// TIA Portal V17 export
// export: Created 2025-06-26T06:49:10.1287295Z, ExportSetting WithDefaults, DisplayName Totally Integrated Automation Portal, DisplayVersion V17 Update 8, DisplayName TIA Portal Openness, DisplayVersion V17 Update 8, DisplayName TIA Portal Version Control Interface, DisplayVersion V17, DisplayName STEP 7 Professional, DisplayVersion V17 Update 8, DisplayName STEP 7 Safety, DisplayVersion V17 Update 6, DisplayName WinCC Advanced, DisplayVersion V17 Update 8
FUNCTION_BLOCK "AnalogInputProcessing"   // FB37, FBD
TITLE = Handle analog inputs
{ S7_Optimized_Access := 'TRUE' }
AUTHOR : Heaten
VERSION : 0.1
// Map & scale analog inputs
// stored: AutoNumber true, IsIECCheckEnabled false, IsRetainMemResEnabled false, MemoryReserve 0, SetENOAutomatically false, UDAEnableTagReadback false
   VAR
      bHere : Bool;
   END_VAR
   VAR_TEMP
      fDummy : Real;
      fMaxWindingTemperature : Real;
      HBL_PT_05 : Real;
   END_VAR
   VAR_TEMP   // added for the SCL form of the ladder/FBD networks
      _w1 : Bool;
   END_VAR
BEGIN

REGION Network 1: HBL_TT_03 Oil sump oil temperature
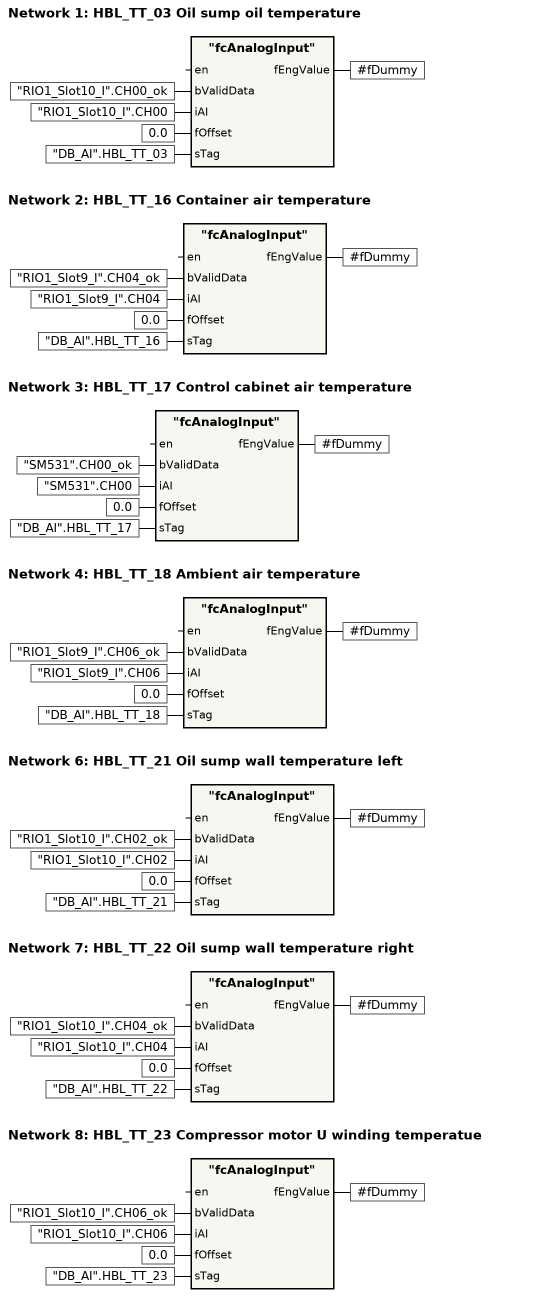
   "fcAnalogInput"(bValidData := "RIO1_Slot10_I".CH00_ok,
                   iAI := "RIO1_Slot10_I".CH00,
                   fOffset := 0.0,
                   sTag := "DB_AI".HBL_TT_03,
                   fEngValue => #fDummy);
END_REGION

REGION Network 2: HBL_TT_16 Container air temperature
   "fcAnalogInput"(bValidData := "RIO1_Slot9_I".CH04_ok,
                   iAI := "RIO1_Slot9_I".CH04,
                   fOffset := 0.0,
                   sTag := "DB_AI".HBL_TT_16,
                   fEngValue => #fDummy);
END_REGION

REGION Network 3: HBL_TT_17 Control cabinet air temperature
   "fcAnalogInput"(bValidData := "SM531".CH00_ok,
                   iAI := "SM531".CH00,
                   fOffset := 0.0,
                   sTag := "DB_AI".HBL_TT_17,
                   fEngValue => #fDummy);
END_REGION

REGION Network 4: HBL_TT_18 Ambient air temperature
   "fcAnalogInput"(bValidData := "RIO1_Slot9_I".CH06_ok,
                   iAI := "RIO1_Slot9_I".CH06,
                   fOffset := 0.0,
                   sTag := "DB_AI".HBL_TT_18,
                   fEngValue => #fDummy);
END_REGION

REGION Network 5: HBL_TT_19 Main inverter temperature
   // ##This is a fieldbus value. get from inverter, if we need it.
END_REGION

REGION Network 6: HBL_TT_21 Oil sump wall temperature left
   "fcAnalogInput"(bValidData := "RIO1_Slot10_I".CH02_ok,
                   iAI := "RIO1_Slot10_I".CH02,
                   fOffset := 0.0,
                   sTag := "DB_AI".HBL_TT_21,
                   fEngValue => #fDummy);
END_REGION

REGION Network 7: HBL_TT_22 Oil sump wall temperature right
   "fcAnalogInput"(bValidData := "RIO1_Slot10_I".CH04_ok,
                   iAI := "RIO1_Slot10_I".CH04,
                   fOffset := 0.0,
                   sTag := "DB_AI".HBL_TT_22,
                   fEngValue => #fDummy);
END_REGION

REGION Network 8: HBL_TT_23 Compressor motor U winding temperatue
   "fcAnalogInput"(bValidData := "RIO1_Slot10_I".CH06_ok,
                   iAI := "RIO1_Slot10_I".CH06,
                   fOffset := 0.0,
                   sTag := "DB_AI".HBL_TT_23,
                   fEngValue => #fDummy);
END_REGION

REGION Network 9: HBL_TT_24 Compressor motor V winding temperature
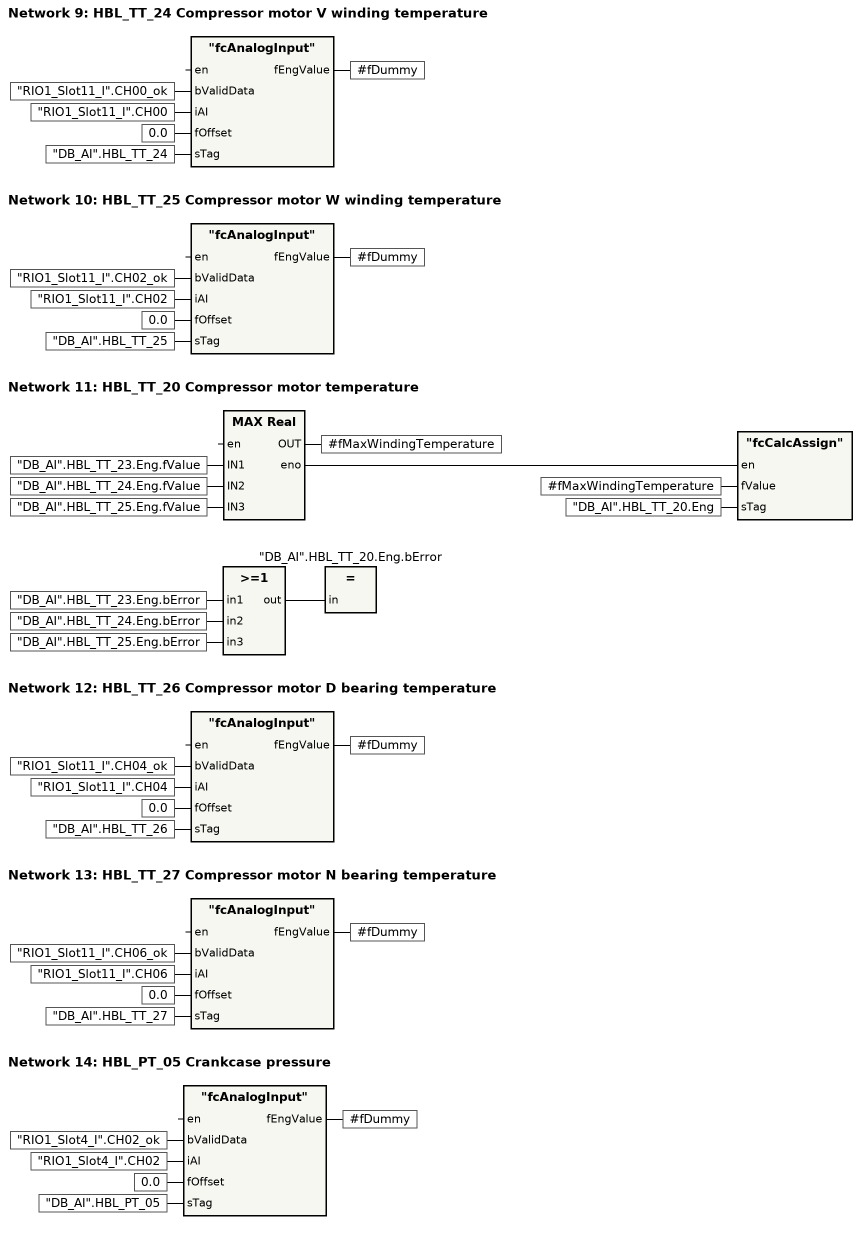
   "fcAnalogInput"(bValidData := "RIO1_Slot11_I".CH00_ok,
                   iAI := "RIO1_Slot11_I".CH00,
                   fOffset := 0.0,
                   sTag := "DB_AI".HBL_TT_24,
                   fEngValue => #fDummy);
END_REGION

REGION Network 10: HBL_TT_25 Compressor motor W winding temperature
   "fcAnalogInput"(bValidData := "RIO1_Slot11_I".CH02_ok,
                   iAI := "RIO1_Slot11_I".CH02,
                   fOffset := 0.0,
                   sTag := "DB_AI".HBL_TT_25,
                   fEngValue => #fDummy);
END_REGION

REGION Network 11: HBL_TT_20 Compressor motor temperature
   // MAX of any of the winding temperatures. If there is only one motor temperature, eg one PTC, use HBL-TT-20 as the analog input object
   // The individual winding temperatures are not used in the program (but are available for monitoring & logging)
   #fMaxWindingTemperature := MAX(IN1 := "DB_AI".HBL_TT_23.Eng.fValue, IN2 := "DB_AI".HBL_TT_24.Eng.fValue, IN3 := "DB_AI".HBL_TT_25.Eng.fValue);
   "fcCalcAssign"(fValue := #fMaxWindingTemperature, sTag := "DB_AI".HBL_TT_20.Eng);
   "DB_AI".HBL_TT_20.Eng.bError := "DB_AI".HBL_TT_23.Eng.bError OR "DB_AI".HBL_TT_24.Eng.bError OR "DB_AI".HBL_TT_25.Eng.bError;
END_REGION

REGION Network 12: HBL_TT_26 Compressor motor D bearing temperature
   "fcAnalogInput"(bValidData := "RIO1_Slot11_I".CH04_ok,
                   iAI := "RIO1_Slot11_I".CH04,
                   fOffset := 0.0,
                   sTag := "DB_AI".HBL_TT_26,
                   fEngValue => #fDummy);
END_REGION

REGION Network 13: HBL_TT_27 Compressor motor N bearing temperature
   "fcAnalogInput"(bValidData := "RIO1_Slot11_I".CH06_ok,
                   iAI := "RIO1_Slot11_I".CH06,
                   fOffset := 0.0,
                   sTag := "DB_AI".HBL_TT_27,
                   fEngValue => #fDummy);
END_REGION

REGION Network 14: HBL_PT_05 Crankcase pressure
   "fcAnalogInput"(bValidData := "RIO1_Slot4_I".CH02_ok,
                   iAI := "RIO1_Slot4_I".CH02,
                   fOffset := 0.0,
                   sTag := "DB_AI".HBL_PT_05,
                   fEngValue => #fDummy);
END_REGION

REGION Network 15: HBL_CT_01 Gas detector
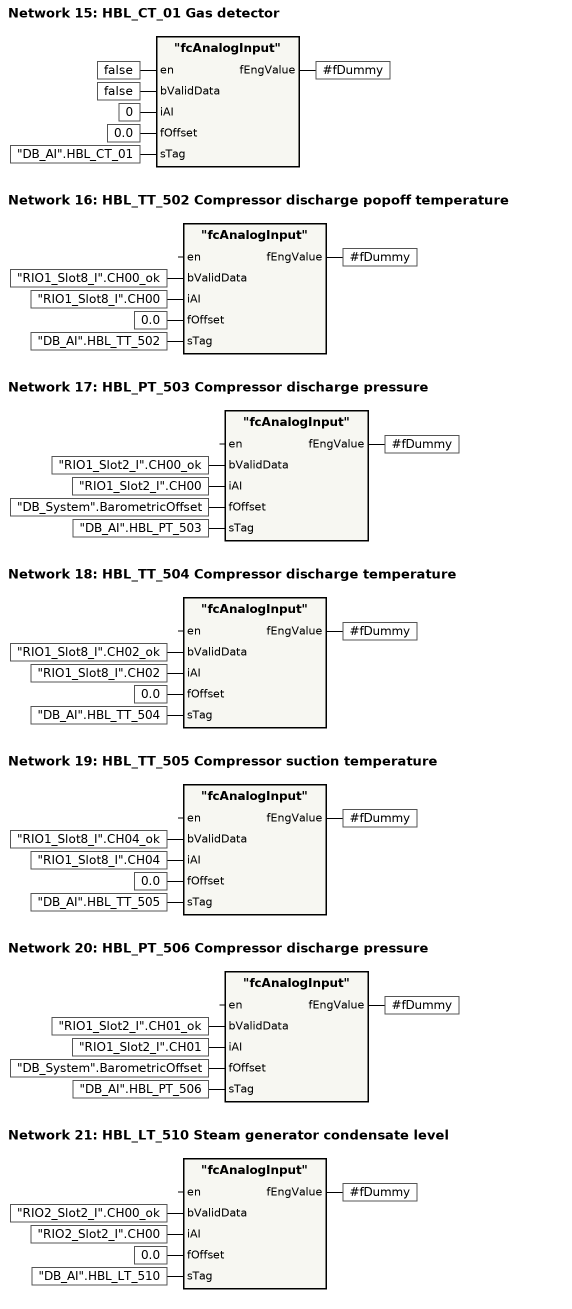
   IF false THEN
       "fcAnalogInput"(bValidData := false,
                       iAI := 0,
                       fOffset := 0.0,
                       sTag := "DB_AI".HBL_CT_01,
                       fEngValue => #fDummy);
   END_IF;
END_REGION

REGION Network 16: HBL_TT_502 Compressor discharge popoff temperature
   "fcAnalogInput"(bValidData := "RIO1_Slot8_I".CH00_ok,
                   iAI := "RIO1_Slot8_I".CH00,
                   fOffset := 0.0,
                   sTag := "DB_AI".HBL_TT_502,
                   fEngValue => #fDummy);
END_REGION

REGION Network 17: HBL_PT_503 Compressor discharge pressure
   "fcAnalogInput"(bValidData := "RIO1_Slot2_I".CH00_ok,
                   iAI := "RIO1_Slot2_I".CH00,
                   fOffset := "DB_System".BarometricOffset,
                   sTag := "DB_AI".HBL_PT_503,
                   fEngValue => #fDummy);
END_REGION

REGION Network 18: HBL_TT_504 Compressor discharge temperature
   "fcAnalogInput"(bValidData := "RIO1_Slot8_I".CH02_ok,
                   iAI := "RIO1_Slot8_I".CH02,
                   fOffset := 0.0,
                   sTag := "DB_AI".HBL_TT_504,
                   fEngValue => #fDummy);
END_REGION

REGION Network 19: HBL_TT_505 Compressor suction temperature
   "fcAnalogInput"(bValidData := "RIO1_Slot8_I".CH04_ok,
                   iAI := "RIO1_Slot8_I".CH04,
                   fOffset := 0.0,
                   sTag := "DB_AI".HBL_TT_505,
                   fEngValue => #fDummy);
END_REGION

REGION Network 20: HBL_PT_506 Compressor discharge pressure
   "fcAnalogInput"(bValidData := "RIO1_Slot2_I".CH01_ok,
                   iAI := "RIO1_Slot2_I".CH01,
                   fOffset := "DB_System".BarometricOffset,
                   sTag := "DB_AI".HBL_PT_506,
                   fEngValue => #fDummy);
END_REGION

REGION Network 21: HBL_LT_510 Steam generator condensate level
   "fcAnalogInput"(bValidData := "RIO2_Slot2_I".CH00_ok,
                   iAI := "RIO2_Slot2_I".CH00,
                   fOffset := 0.0,
                   sTag := "DB_AI".HBL_LT_510,
                   fEngValue => #fDummy);
END_REGION

REGION Network 22: HBL_PT_511 Heat sink discharge pressure
   // Local or remote
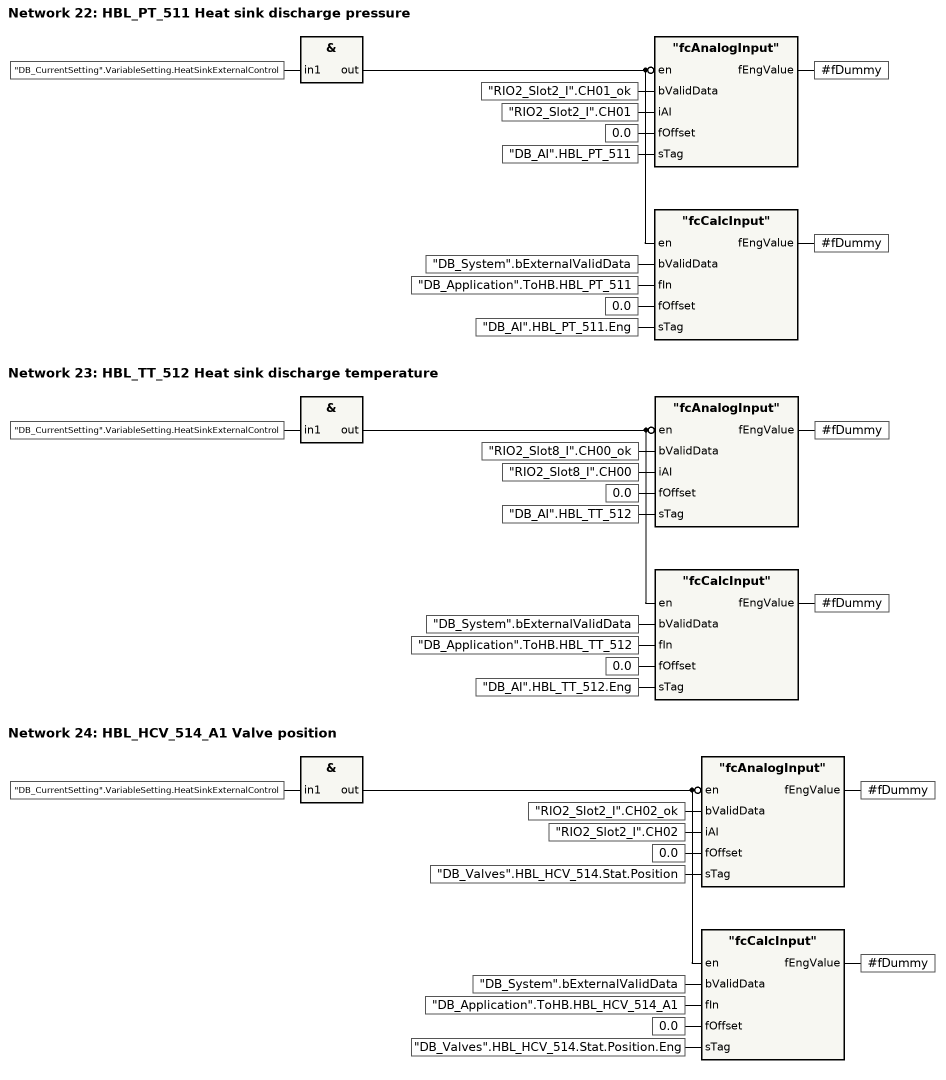
   #_w1 := "DB_CurrentSetting".VariableSetting.HeatSinkExternalControl;
   IF NOT "DB_CurrentSetting".VariableSetting.HeatSinkExternalControl THEN
       "fcAnalogInput"(bValidData := "RIO2_Slot2_I".CH01_ok,
                       iAI := "RIO2_Slot2_I".CH01,
                       fOffset := 0.0,
                       sTag := "DB_AI".HBL_PT_511,
                       fEngValue => #fDummy);
   END_IF;
   IF #_w1 THEN
       "fcCalcInput"(bValidData := "DB_System".bExternalValidData,
                     fIn := "DB_Application".ToHB.HBL_PT_511,
                     fOffset := 0.0,
                     sTag := "DB_AI".HBL_PT_511.Eng,
                     fEngValue => #fDummy);
   END_IF;
END_REGION

REGION Network 23: HBL_TT_512 Heat sink discharge temperature
   // Local or remote
   #_w1 := "DB_CurrentSetting".VariableSetting.HeatSinkExternalControl;
   IF NOT "DB_CurrentSetting".VariableSetting.HeatSinkExternalControl THEN
       "fcAnalogInput"(bValidData := "RIO2_Slot8_I".CH00_ok,
                       iAI := "RIO2_Slot8_I".CH00,
                       fOffset := 0.0,
                       sTag := "DB_AI".HBL_TT_512,
                       fEngValue => #fDummy);
   END_IF;
   IF #_w1 THEN
       "fcCalcInput"(bValidData := "DB_System".bExternalValidData,
                     fIn := "DB_Application".ToHB.HBL_TT_512,
                     fOffset := 0.0,
                     sTag := "DB_AI".HBL_TT_512.Eng,
                     fEngValue => #fDummy);
   END_IF;
END_REGION

REGION Network 24: HBL_HCV_514_A1 Valve position
   // Local or remote
   #_w1 := "DB_CurrentSetting".VariableSetting.HeatSinkExternalControl;
   IF NOT "DB_CurrentSetting".VariableSetting.HeatSinkExternalControl THEN
       "fcAnalogInput"(bValidData := "RIO2_Slot2_I".CH02_ok,
                       iAI := "RIO2_Slot2_I".CH02,
                       fOffset := 0.0,
                       sTag := "DB_Valves".HBL_HCV_514.Stat.Position,
                       fEngValue => #fDummy);
   END_IF;
   IF #_w1 THEN
       "fcCalcInput"(bValidData := "DB_System".bExternalValidData,
                     fIn := "DB_Application".ToHB.HBL_HCV_514_A1,
                     fOffset := 0.0,
                     sTag := "DB_Valves".HBL_HCV_514.Stat.Position.Eng,
                     fEngValue => #fDummy);
   END_IF;
END_REGION

REGION Network 25: HBL_HCV_515_A1 Heat sink condensate blowdown valve position
   // Local or remote
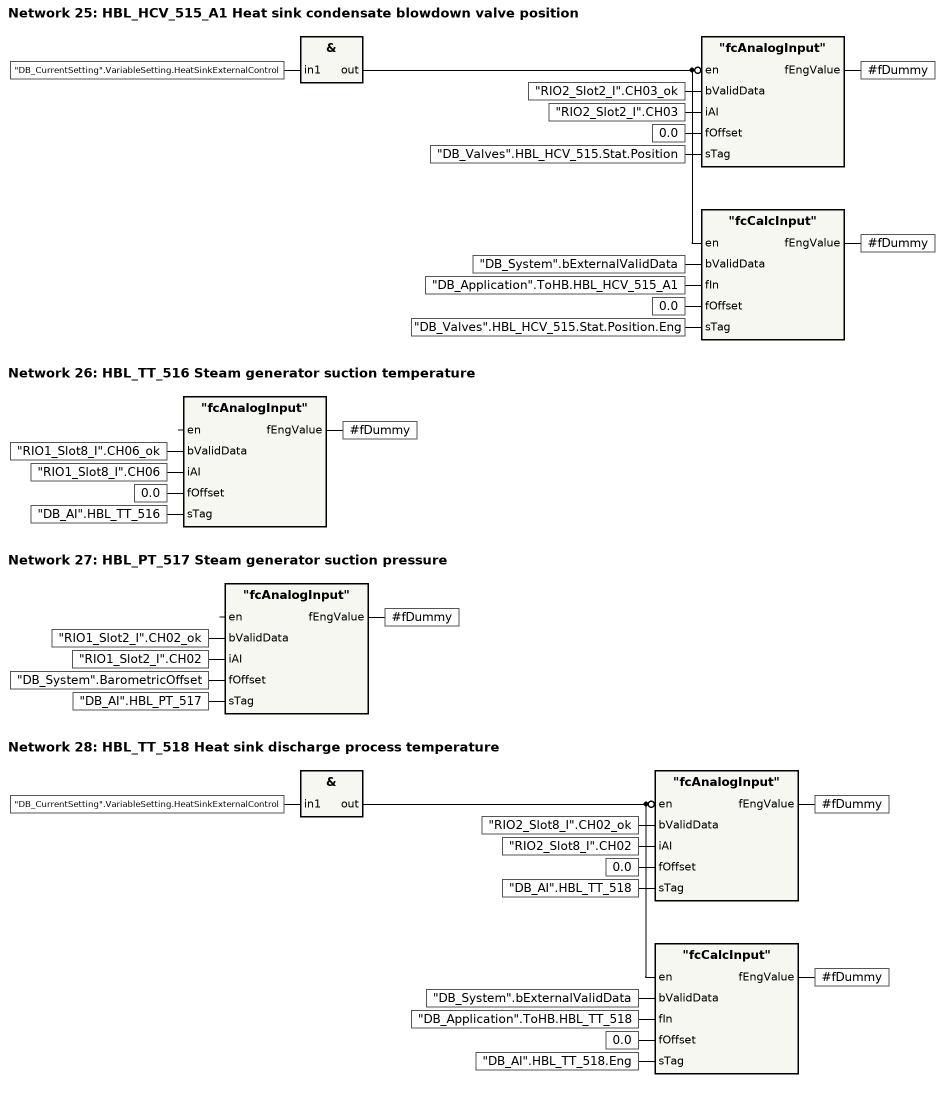
   #_w1 := "DB_CurrentSetting".VariableSetting.HeatSinkExternalControl;
   IF NOT "DB_CurrentSetting".VariableSetting.HeatSinkExternalControl THEN
       "fcAnalogInput"(bValidData := "RIO2_Slot2_I".CH03_ok,
                       iAI := "RIO2_Slot2_I".CH03,
                       fOffset := 0.0,
                       sTag := "DB_Valves".HBL_HCV_515.Stat.Position,
                       fEngValue => #fDummy);
   END_IF;
   IF #_w1 THEN
       "fcCalcInput"(bValidData := "DB_System".bExternalValidData,
                     fIn := "DB_Application".ToHB.HBL_HCV_515_A1,
                     fOffset := 0.0,
                     sTag := "DB_Valves".HBL_HCV_515.Stat.Position.Eng,
                     fEngValue => #fDummy);
   END_IF;
END_REGION

REGION Network 26: HBL_TT_516 Steam generator suction temperature
   "fcAnalogInput"(bValidData := "RIO1_Slot8_I".CH06_ok,
                   iAI := "RIO1_Slot8_I".CH06,
                   fOffset := 0.0,
                   sTag := "DB_AI".HBL_TT_516,
                   fEngValue => #fDummy);
END_REGION

REGION Network 27: HBL_PT_517 Steam generator suction pressure
   "fcAnalogInput"(bValidData := "RIO1_Slot2_I".CH02_ok,
                   iAI := "RIO1_Slot2_I".CH02,
                   fOffset := "DB_System".BarometricOffset,
                   sTag := "DB_AI".HBL_PT_517,
                   fEngValue => #fDummy);
END_REGION

REGION Network 28: HBL_TT_518 Heat sink discharge process temperature
   // Local or remote
   #_w1 := "DB_CurrentSetting".VariableSetting.HeatSinkExternalControl;
   IF NOT "DB_CurrentSetting".VariableSetting.HeatSinkExternalControl THEN
       "fcAnalogInput"(bValidData := "RIO2_Slot8_I".CH02_ok,
                       iAI := "RIO2_Slot8_I".CH02,
                       fOffset := 0.0,
                       sTag := "DB_AI".HBL_TT_518,
                       fEngValue => #fDummy);
   END_IF;
   IF #_w1 THEN
       "fcCalcInput"(bValidData := "DB_System".bExternalValidData,
                     fIn := "DB_Application".ToHB.HBL_TT_518,
                     fOffset := 0.0,
                     sTag := "DB_AI".HBL_TT_518.Eng,
                     fEngValue => #fDummy);
   END_IF;
END_REGION

REGION Network 29: HBL_PT_519 Heat sink discharge process pressure
   // Local or remote
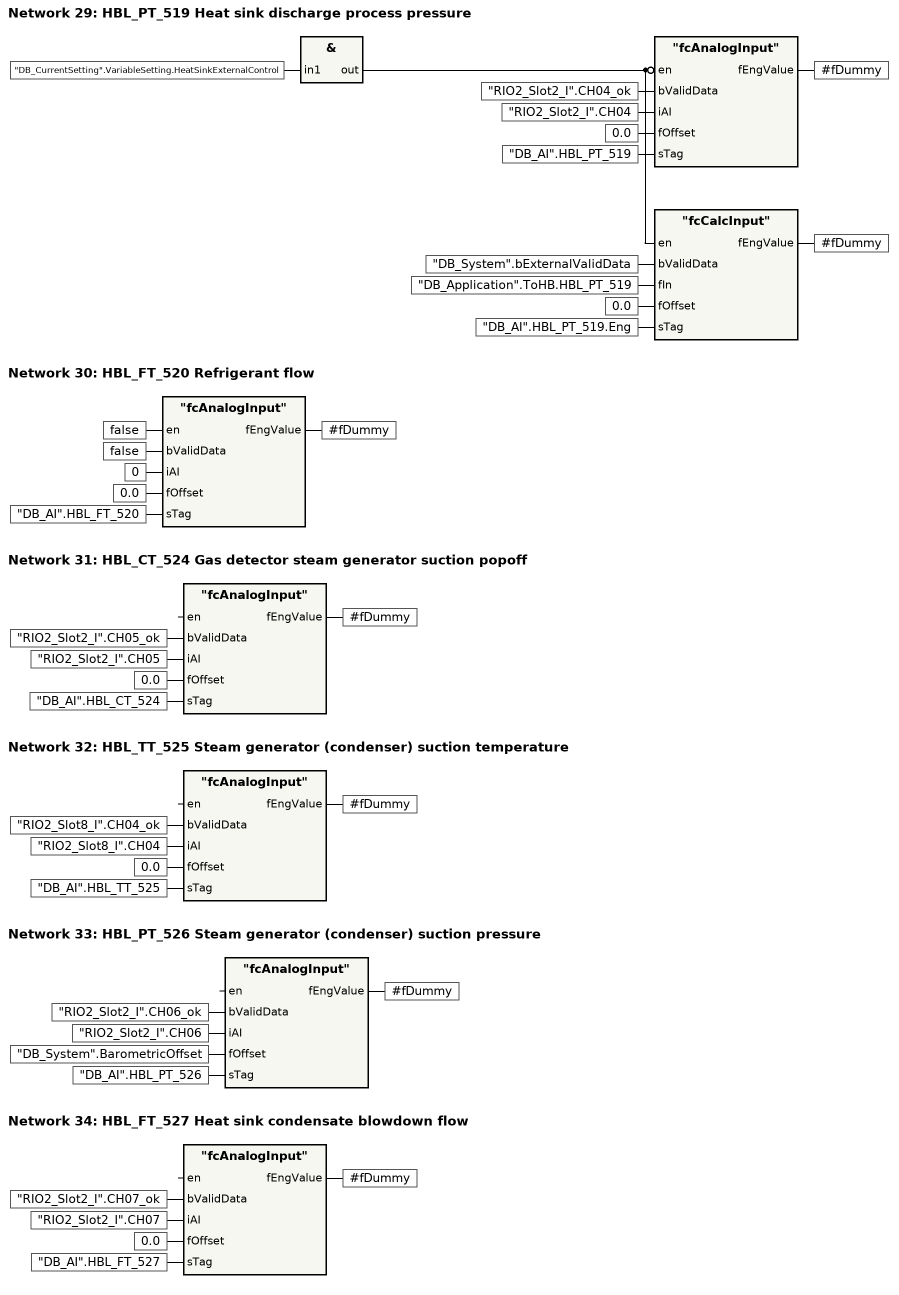
   #_w1 := "DB_CurrentSetting".VariableSetting.HeatSinkExternalControl;
   IF NOT "DB_CurrentSetting".VariableSetting.HeatSinkExternalControl THEN
       "fcAnalogInput"(bValidData := "RIO2_Slot2_I".CH04_ok,
                       iAI := "RIO2_Slot2_I".CH04,
                       fOffset := 0.0,
                       sTag := "DB_AI".HBL_PT_519,
                       fEngValue => #fDummy);
   END_IF;
   IF #_w1 THEN
       "fcCalcInput"(bValidData := "DB_System".bExternalValidData,
                     fIn := "DB_Application".ToHB.HBL_PT_519,
                     fOffset := 0.0,
                     sTag := "DB_AI".HBL_PT_519.Eng,
                     fEngValue => #fDummy);
   END_IF;
END_REGION

REGION Network 30: HBL_FT_520 Refrigerant flow
   // Not used in Offenau
   IF false THEN
       "fcAnalogInput"(bValidData := false,
                       iAI := 0,
                       fOffset := 0.0,
                       sTag := "DB_AI".HBL_FT_520,
                       fEngValue => #fDummy);
   END_IF;
END_REGION

REGION Network 31: HBL_CT_524 Gas detector steam generator suction popoff
   "fcAnalogInput"(bValidData := "RIO2_Slot2_I".CH05_ok,
                   iAI := "RIO2_Slot2_I".CH05,
                   fOffset := 0.0,
                   sTag := "DB_AI".HBL_CT_524,
                   fEngValue => #fDummy);
END_REGION

REGION Network 32: HBL_TT_525 Steam generator (condenser) suction temperature
   "fcAnalogInput"(bValidData := "RIO2_Slot8_I".CH04_ok,
                   iAI := "RIO2_Slot8_I".CH04,
                   fOffset := 0.0,
                   sTag := "DB_AI".HBL_TT_525,
                   fEngValue => #fDummy);
END_REGION

REGION Network 33: HBL_PT_526 Steam generator (condenser) suction pressure
   "fcAnalogInput"(bValidData := "RIO2_Slot2_I".CH06_ok,
                   iAI := "RIO2_Slot2_I".CH06,
                   fOffset := "DB_System".BarometricOffset,
                   sTag := "DB_AI".HBL_PT_526,
                   fEngValue => #fDummy);
END_REGION

REGION Network 34: HBL_FT_527 Heat sink condensate blowdown flow
   "fcAnalogInput"(bValidData := "RIO2_Slot2_I".CH07_ok,
                   iAI := "RIO2_Slot2_I".CH07,
                   fOffset := 0.0,
                   sTag := "DB_AI".HBL_FT_527,
                   fEngValue => #fDummy);
END_REGION

REGION Network 35: HBL_TT_530 Expansion valve B discharge temperature
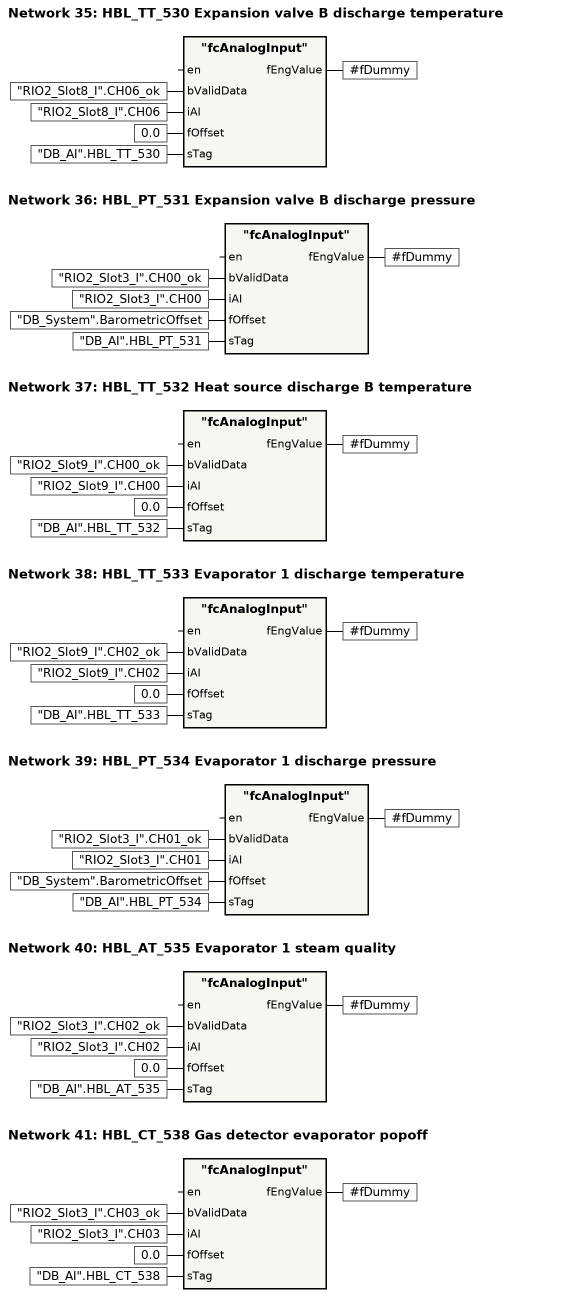
   "fcAnalogInput"(bValidData := "RIO2_Slot8_I".CH06_ok,
                   iAI := "RIO2_Slot8_I".CH06,
                   fOffset := 0.0,
                   sTag := "DB_AI".HBL_TT_530,
                   fEngValue => #fDummy);
END_REGION

REGION Network 36: HBL_PT_531 Expansion valve B discharge pressure
   // Convert from rel to abs
   "fcAnalogInput"(bValidData := "RIO2_Slot3_I".CH00_ok,
                   iAI := "RIO2_Slot3_I".CH00,
                   fOffset := "DB_System".BarometricOffset,
                   sTag := "DB_AI".HBL_PT_531,
                   fEngValue => #fDummy);
END_REGION

REGION Network 37: HBL_TT_532 Heat source discharge B temperature
   "fcAnalogInput"(bValidData := "RIO2_Slot9_I".CH00_ok,
                   iAI := "RIO2_Slot9_I".CH00,
                   fOffset := 0.0,
                   sTag := "DB_AI".HBL_TT_532,
                   fEngValue => #fDummy);
END_REGION

REGION Network 38: HBL_TT_533 Evaporator 1 discharge temperature
   "fcAnalogInput"(bValidData := "RIO2_Slot9_I".CH02_ok,
                   iAI := "RIO2_Slot9_I".CH02,
                   fOffset := 0.0,
                   sTag := "DB_AI".HBL_TT_533,
                   fEngValue => #fDummy);
END_REGION

REGION Network 39: HBL_PT_534 Evaporator 1 discharge pressure
   // Convert from rel to abs
   "fcAnalogInput"(bValidData := "RIO2_Slot3_I".CH01_ok,
                   iAI := "RIO2_Slot3_I".CH01,
                   fOffset := "DB_System".BarometricOffset,
                   sTag := "DB_AI".HBL_PT_534,
                   fEngValue => #fDummy);
END_REGION

REGION Network 40: HBL_AT_535 Evaporator 1 steam quality
   "fcAnalogInput"(bValidData := "RIO2_Slot3_I".CH02_ok,
                   iAI := "RIO2_Slot3_I".CH02,
                   fOffset := 0.0,
                   sTag := "DB_AI".HBL_AT_535,
                   fEngValue => #fDummy);
END_REGION

REGION Network 41: HBL_CT_538 Gas detector evaporator popoff
   "fcAnalogInput"(bValidData := "RIO2_Slot3_I".CH03_ok,
                   iAI := "RIO2_Slot3_I".CH03,
                   fOffset := 0.0,
                   sTag := "DB_AI".HBL_CT_538,
                   fEngValue => #fDummy);
END_REGION

REGION Network 42: HBL_TT_540 Expansion valve A discharge temperature
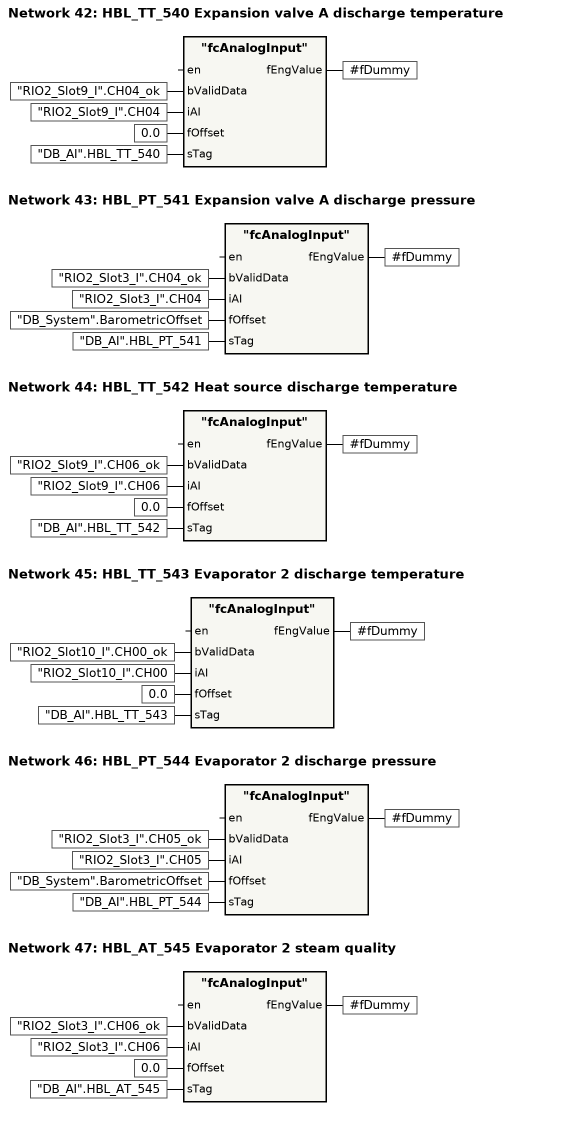
   "fcAnalogInput"(bValidData := "RIO2_Slot9_I".CH04_ok,
                   iAI := "RIO2_Slot9_I".CH04,
                   fOffset := 0.0,
                   sTag := "DB_AI".HBL_TT_540,
                   fEngValue => #fDummy);
END_REGION

REGION Network 43: HBL_PT_541 Expansion valve A discharge pressure
   "fcAnalogInput"(bValidData := "RIO2_Slot3_I".CH04_ok,
                   iAI := "RIO2_Slot3_I".CH04,
                   fOffset := "DB_System".BarometricOffset,
                   sTag := "DB_AI".HBL_PT_541,
                   fEngValue => #fDummy);
END_REGION

REGION Network 44: HBL_TT_542 Heat source discharge temperature
   "fcAnalogInput"(bValidData := "RIO2_Slot9_I".CH06_ok,
                   iAI := "RIO2_Slot9_I".CH06,
                   fOffset := 0.0,
                   sTag := "DB_AI".HBL_TT_542,
                   fEngValue => #fDummy);
END_REGION

REGION Network 45: HBL_TT_543 Evaporator 2 discharge temperature
   "fcAnalogInput"(bValidData := "RIO2_Slot10_I".CH00_ok,
                   iAI := "RIO2_Slot10_I".CH00,
                   fOffset := 0.0,
                   sTag := "DB_AI".HBL_TT_543,
                   fEngValue => #fDummy);
END_REGION

REGION Network 46: HBL_PT_544 Evaporator 2 discharge pressure
   "fcAnalogInput"(bValidData := "RIO2_Slot3_I".CH05_ok,
                   iAI := "RIO2_Slot3_I".CH05,
                   fOffset := "DB_System".BarometricOffset,
                   sTag := "DB_AI".HBL_PT_544,
                   fEngValue => #fDummy);
END_REGION

REGION Network 47: HBL_AT_545 Evaporator 2 steam quality
   "fcAnalogInput"(bValidData := "RIO2_Slot3_I".CH06_ok,
                   iAI := "RIO2_Slot3_I".CH06,
                   fOffset := 0.0,
                   sTag := "DB_AI".HBL_AT_545,
                   fEngValue => #fDummy);
END_REGION

REGION Network 48: HBL_TT_546 Heat source suction temperature
   // Local or remote
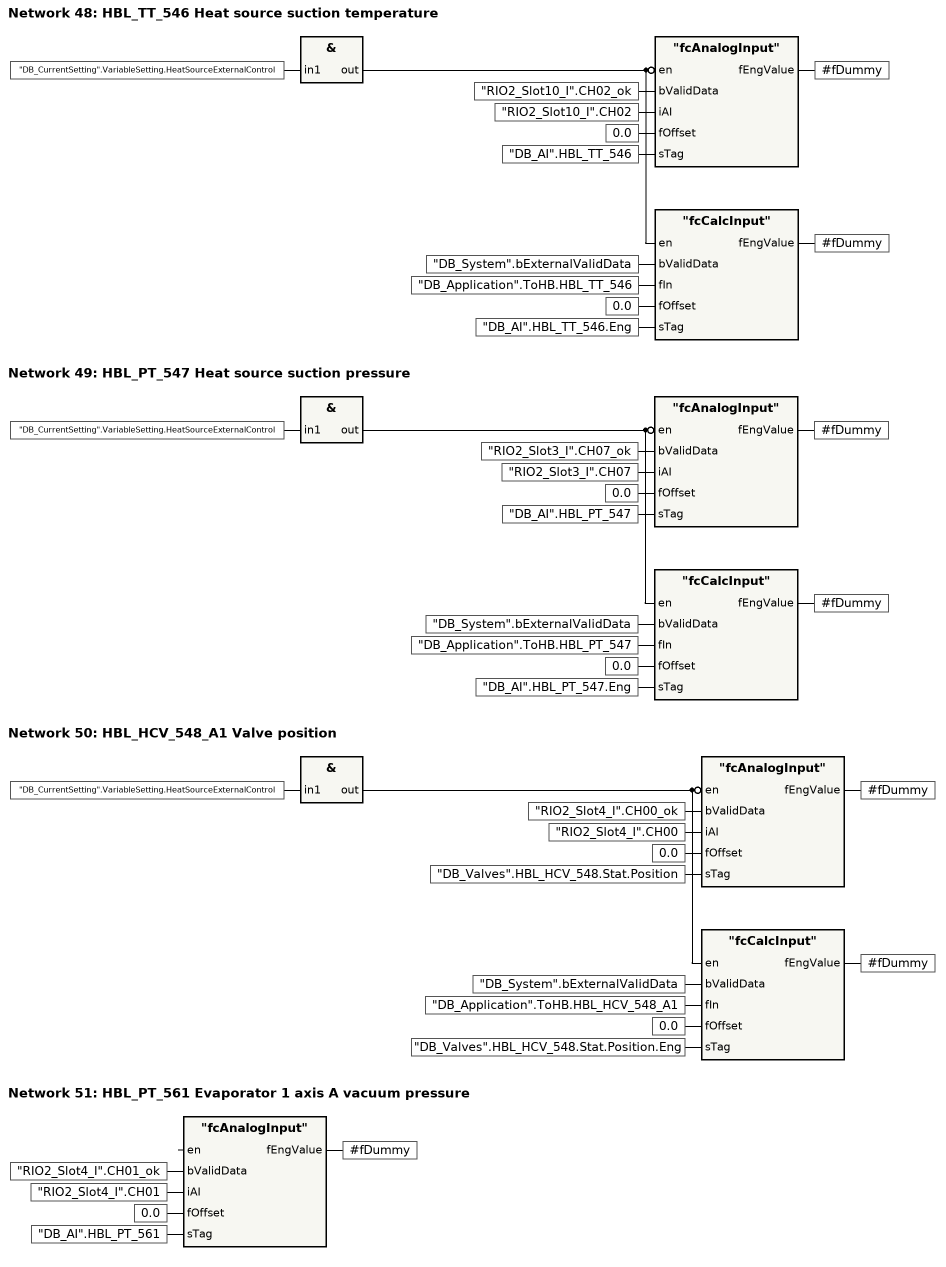
   #_w1 := "DB_CurrentSetting".VariableSetting.HeatSourceExternalControl;
   IF NOT "DB_CurrentSetting".VariableSetting.HeatSourceExternalControl THEN
       "fcAnalogInput"(bValidData := "RIO2_Slot10_I".CH02_ok,
                       iAI := "RIO2_Slot10_I".CH02,
                       fOffset := 0.0,
                       sTag := "DB_AI".HBL_TT_546,
                       fEngValue => #fDummy);
   END_IF;
   IF #_w1 THEN
       "fcCalcInput"(bValidData := "DB_System".bExternalValidData,
                     fIn := "DB_Application".ToHB.HBL_TT_546,
                     fOffset := 0.0,
                     sTag := "DB_AI".HBL_TT_546.Eng,
                     fEngValue => #fDummy);
   END_IF;
END_REGION

REGION Network 49: HBL_PT_547 Heat source suction pressure
   // Local or remote
   #_w1 := "DB_CurrentSetting".VariableSetting.HeatSourceExternalControl;
   IF NOT "DB_CurrentSetting".VariableSetting.HeatSourceExternalControl THEN
       "fcAnalogInput"(bValidData := "RIO2_Slot3_I".CH07_ok,
                       iAI := "RIO2_Slot3_I".CH07,
                       fOffset := 0.0,
                       sTag := "DB_AI".HBL_PT_547,
                       fEngValue => #fDummy);
   END_IF;
   IF #_w1 THEN
       "fcCalcInput"(bValidData := "DB_System".bExternalValidData,
                     fIn := "DB_Application".ToHB.HBL_PT_547,
                     fOffset := 0.0,
                     sTag := "DB_AI".HBL_PT_547.Eng,
                     fEngValue => #fDummy);
   END_IF;
END_REGION

REGION Network 50: HBL_HCV_548_A1 Valve position
   // Local or remote
   #_w1 := "DB_CurrentSetting".VariableSetting.HeatSourceExternalControl;
   IF NOT "DB_CurrentSetting".VariableSetting.HeatSourceExternalControl THEN
       "fcAnalogInput"(bValidData := "RIO2_Slot4_I".CH00_ok,
                       iAI := "RIO2_Slot4_I".CH00,
                       fOffset := 0.0,
                       sTag := "DB_Valves".HBL_HCV_548.Stat.Position,
                       fEngValue => #fDummy);
   END_IF;
   IF #_w1 THEN
       "fcCalcInput"(bValidData := "DB_System".bExternalValidData,
                     fIn := "DB_Application".ToHB.HBL_HCV_548_A1,
                     fOffset := 0.0,
                     sTag := "DB_Valves".HBL_HCV_548.Stat.Position.Eng,
                     fEngValue => #fDummy);
   END_IF;
END_REGION

REGION Network 51: HBL_PT_561 Evaporator 1 axis A vacuum pressure
   "fcAnalogInput"(bValidData := "RIO2_Slot4_I".CH01_ok,
                   iAI := "RIO2_Slot4_I".CH01,
                   fOffset := 0.0,
                   sTag := "DB_AI".HBL_PT_561,
                   fEngValue => #fDummy);
END_REGION

REGION Network 52: HBL_PT_562 Evaporator 2 axis A vacuum pressure
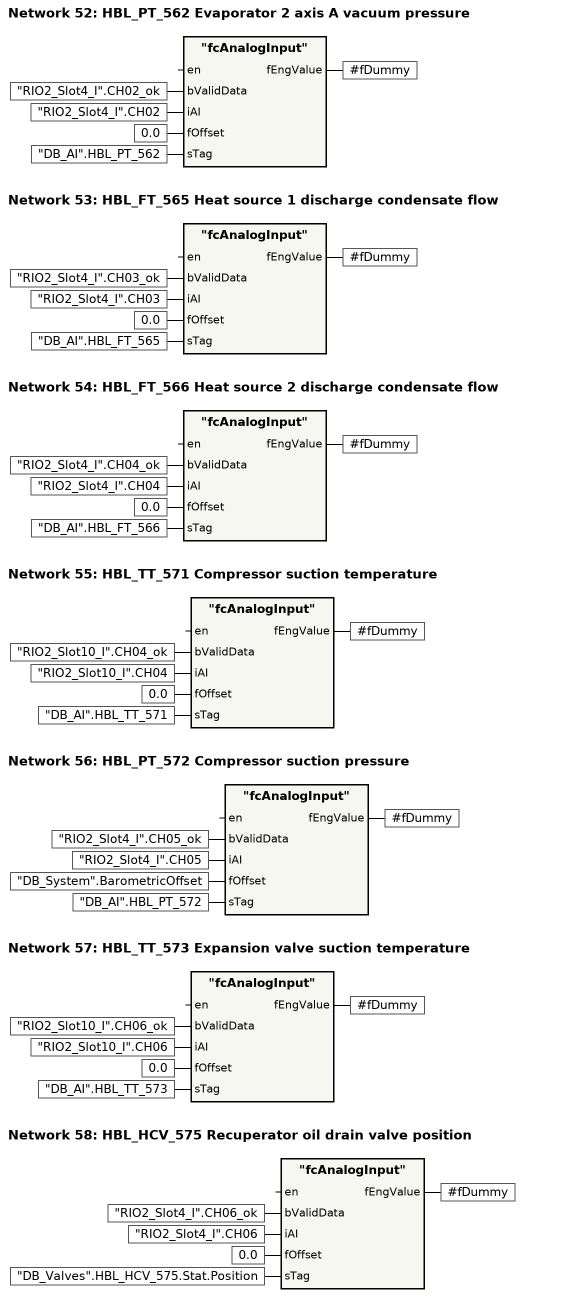
   "fcAnalogInput"(bValidData := "RIO2_Slot4_I".CH02_ok,
                   iAI := "RIO2_Slot4_I".CH02,
                   fOffset := 0.0,
                   sTag := "DB_AI".HBL_PT_562,
                   fEngValue => #fDummy);
END_REGION

REGION Network 53: HBL_FT_565 Heat source 1 discharge condensate flow
   "fcAnalogInput"(bValidData := "RIO2_Slot4_I".CH03_ok,
                   iAI := "RIO2_Slot4_I".CH03,
                   fOffset := 0.0,
                   sTag := "DB_AI".HBL_FT_565,
                   fEngValue => #fDummy);
END_REGION

REGION Network 54: HBL_FT_566 Heat source 2 discharge condensate flow
   "fcAnalogInput"(bValidData := "RIO2_Slot4_I".CH04_ok,
                   iAI := "RIO2_Slot4_I".CH04,
                   fOffset := 0.0,
                   sTag := "DB_AI".HBL_FT_566,
                   fEngValue => #fDummy);
END_REGION

REGION Network 55: HBL_TT_571 Compressor suction temperature
   "fcAnalogInput"(bValidData := "RIO2_Slot10_I".CH04_ok,
                   iAI := "RIO2_Slot10_I".CH04,
                   fOffset := 0.0,
                   sTag := "DB_AI".HBL_TT_571,
                   fEngValue => #fDummy);
END_REGION

REGION Network 56: HBL_PT_572 Compressor suction pressure
   "fcAnalogInput"(bValidData := "RIO2_Slot4_I".CH05_ok,
                   iAI := "RIO2_Slot4_I".CH05,
                   fOffset := "DB_System".BarometricOffset,
                   sTag := "DB_AI".HBL_PT_572,
                   fEngValue => #fDummy);
END_REGION

REGION Network 57: HBL_TT_573 Expansion valve suction temperature
   "fcAnalogInput"(bValidData := "RIO2_Slot10_I".CH06_ok,
                   iAI := "RIO2_Slot10_I".CH06,
                   fOffset := 0.0,
                   sTag := "DB_AI".HBL_TT_573,
                   fEngValue => #fDummy);
END_REGION

REGION Network 58: HBL_HCV_575 Recuperator oil drain valve position
   "fcAnalogInput"(bValidData := "RIO2_Slot4_I".CH06_ok,
                   iAI := "RIO2_Slot4_I".CH06,
                   fOffset := 0.0,
                   sTag := "DB_Valves".HBL_HCV_575.Stat.Position,
                   fEngValue => #fDummy);
END_REGION

REGION Network 59: HBL_HCV_576 Expansion Valve A position
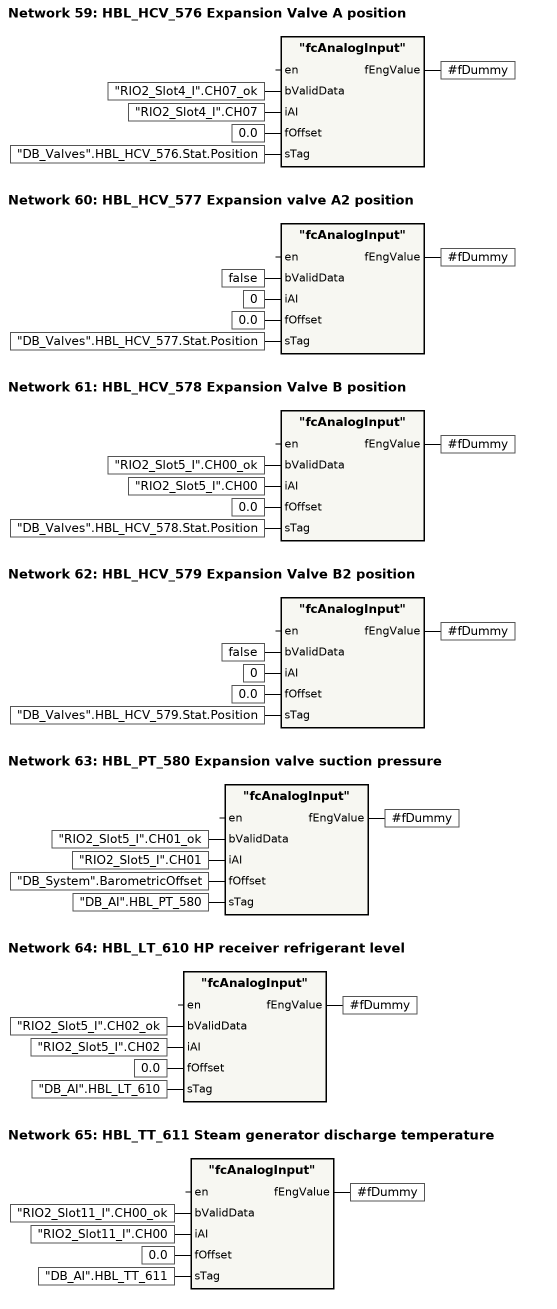
   "fcAnalogInput"(bValidData := "RIO2_Slot4_I".CH07_ok,
                   iAI := "RIO2_Slot4_I".CH07,
                   fOffset := 0.0,
                   sTag := "DB_Valves".HBL_HCV_576.Stat.Position,
                   fEngValue => #fDummy);
END_REGION

REGION Network 60: HBL_HCV_577 Expansion valve A2 position
   "fcAnalogInput"(bValidData := false,
                   iAI := 0,
                   fOffset := 0.0,
                   sTag := "DB_Valves".HBL_HCV_577.Stat.Position,
                   fEngValue => #fDummy);
END_REGION

REGION Network 61: HBL_HCV_578 Expansion Valve B position
   "fcAnalogInput"(bValidData := "RIO2_Slot5_I".CH00_ok,
                   iAI := "RIO2_Slot5_I".CH00,
                   fOffset := 0.0,
                   sTag := "DB_Valves".HBL_HCV_578.Stat.Position,
                   fEngValue => #fDummy);
END_REGION

REGION Network 62: HBL_HCV_579 Expansion Valve B2 position
   "fcAnalogInput"(bValidData := false,
                   iAI := 0,
                   fOffset := 0.0,
                   sTag := "DB_Valves".HBL_HCV_579.Stat.Position,
                   fEngValue => #fDummy);
END_REGION

REGION Network 63: HBL_PT_580 Expansion valve suction pressure
   "fcAnalogInput"(bValidData := "RIO2_Slot5_I".CH01_ok,
                   iAI := "RIO2_Slot5_I".CH01,
                   fOffset := "DB_System".BarometricOffset,
                   sTag := "DB_AI".HBL_PT_580,
                   fEngValue => #fDummy);
END_REGION

REGION Network 64: HBL_LT_610 HP receiver refrigerant level
   "fcAnalogInput"(bValidData := "RIO2_Slot5_I".CH02_ok,
                   iAI := "RIO2_Slot5_I".CH02,
                   fOffset := 0.0,
                   sTag := "DB_AI".HBL_LT_610,
                   fEngValue => #fDummy);
END_REGION

REGION Network 65: HBL_TT_611 Steam generator discharge temperature
   "fcAnalogInput"(bValidData := "RIO2_Slot11_I".CH00_ok,
                   iAI := "RIO2_Slot11_I".CH00,
                   fOffset := 0.0,
                   sTag := "DB_AI".HBL_TT_611,
                   fEngValue => #fDummy);
END_REGION

REGION Network 66: HBL_PT_612 Steam generator discharge pressure
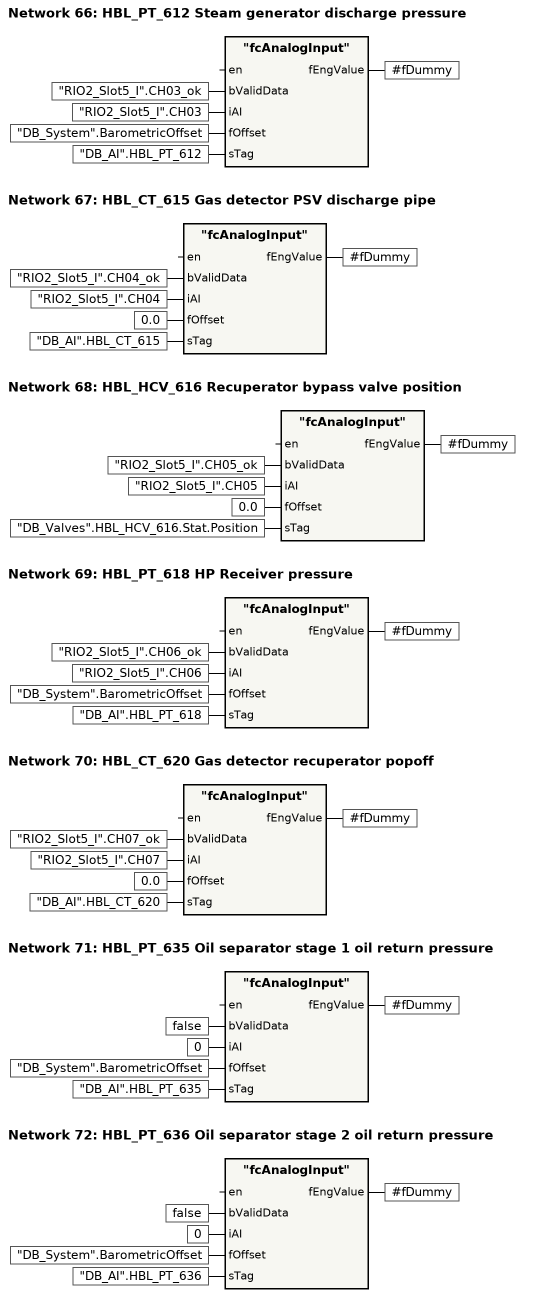
   "fcAnalogInput"(bValidData := "RIO2_Slot5_I".CH03_ok,
                   iAI := "RIO2_Slot5_I".CH03,
                   fOffset := "DB_System".BarometricOffset,
                   sTag := "DB_AI".HBL_PT_612,
                   fEngValue => #fDummy);
END_REGION

REGION Network 67: HBL_CT_615 Gas detector PSV discharge pipe
   "fcAnalogInput"(bValidData := "RIO2_Slot5_I".CH04_ok,
                   iAI := "RIO2_Slot5_I".CH04,
                   fOffset := 0.0,
                   sTag := "DB_AI".HBL_CT_615,
                   fEngValue => #fDummy);
END_REGION

REGION Network 68: HBL_HCV_616 Recuperator bypass valve position
   "fcAnalogInput"(bValidData := "RIO2_Slot5_I".CH05_ok,
                   iAI := "RIO2_Slot5_I".CH05,
                   fOffset := 0.0,
                   sTag := "DB_Valves".HBL_HCV_616.Stat.Position,
                   fEngValue => #fDummy);
END_REGION

REGION Network 69: HBL_PT_618 HP Receiver pressure
   "fcAnalogInput"(bValidData := "RIO2_Slot5_I".CH06_ok,
                   iAI := "RIO2_Slot5_I".CH06,
                   fOffset := "DB_System".BarometricOffset,
                   sTag := "DB_AI".HBL_PT_618,
                   fEngValue => #fDummy);
END_REGION

REGION Network 70: HBL_CT_620 Gas detector recuperator popoff
   "fcAnalogInput"(bValidData := "RIO2_Slot5_I".CH07_ok,
                   iAI := "RIO2_Slot5_I".CH07,
                   fOffset := 0.0,
                   sTag := "DB_AI".HBL_CT_620,
                   fEngValue => #fDummy);
END_REGION

REGION Network 71: HBL_PT_635 Oil separator stage 1 oil return pressure
   "fcAnalogInput"(bValidData := false,
                   iAI := 0,
                   fOffset := "DB_System".BarometricOffset,
                   sTag := "DB_AI".HBL_PT_635,
                   fEngValue => #fDummy);
END_REGION

REGION Network 72: HBL_PT_636 Oil separator stage 2 oil return pressure
   "fcAnalogInput"(bValidData := false,
                   iAI := 0,
                   fOffset := "DB_System".BarometricOffset,
                   sTag := "DB_AI".HBL_PT_636,
                   fEngValue => #fDummy);
END_REGION

REGION Network 73: HBL_CT_643 Gas detector suction accumulator popoff
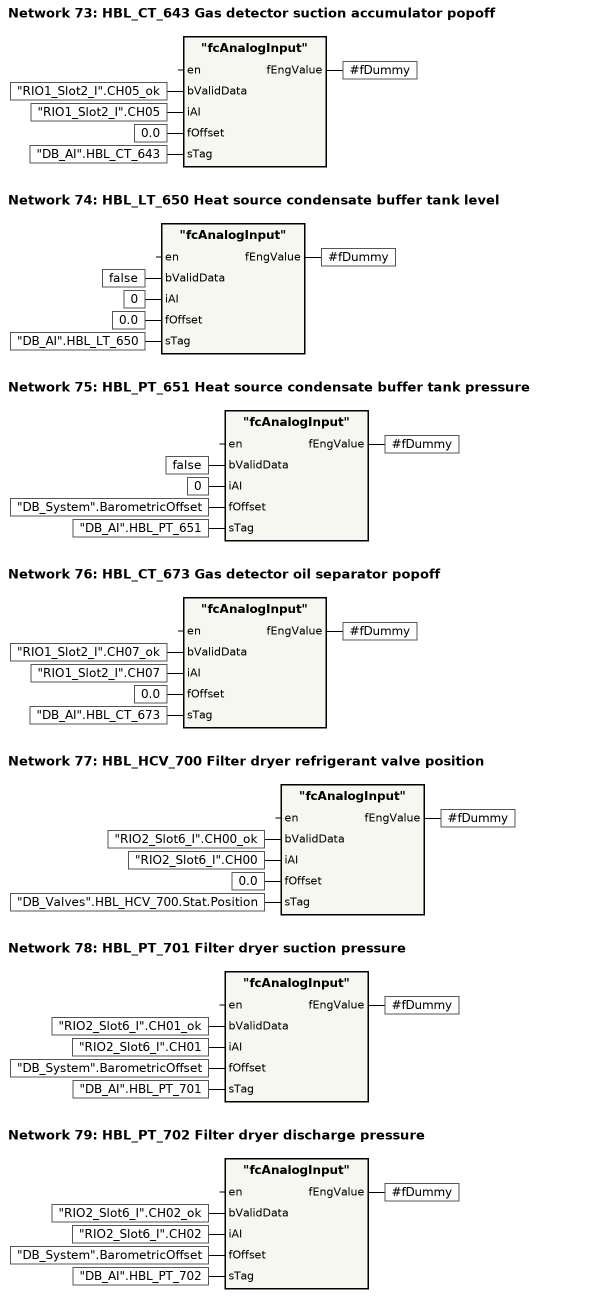
   "fcAnalogInput"(bValidData := "RIO1_Slot2_I".CH05_ok,
                   iAI := "RIO1_Slot2_I".CH05,
                   fOffset := 0.0,
                   sTag := "DB_AI".HBL_CT_643,
                   fEngValue => #fDummy);
END_REGION

REGION Network 74: HBL_LT_650 Heat source condensate buffer tank level
   "fcAnalogInput"(bValidData := false,
                   iAI := 0,
                   fOffset := 0.0,
                   sTag := "DB_AI".HBL_LT_650,
                   fEngValue => #fDummy);
END_REGION

REGION Network 75: HBL_PT_651 Heat source condensate buffer tank pressure
   "fcAnalogInput"(bValidData := false,
                   iAI := 0,
                   fOffset := "DB_System".BarometricOffset,
                   sTag := "DB_AI".HBL_PT_651,
                   fEngValue => #fDummy);
END_REGION

REGION Network 76: HBL_CT_673 Gas detector oil separator popoff
   "fcAnalogInput"(bValidData := "RIO1_Slot2_I".CH07_ok,
                   iAI := "RIO1_Slot2_I".CH07,
                   fOffset := 0.0,
                   sTag := "DB_AI".HBL_CT_673,
                   fEngValue => #fDummy);
END_REGION

REGION Network 77: HBL_HCV_700 Filter dryer refrigerant valve position
   "fcAnalogInput"(bValidData := "RIO2_Slot6_I".CH00_ok,
                   iAI := "RIO2_Slot6_I".CH00,
                   fOffset := 0.0,
                   sTag := "DB_Valves".HBL_HCV_700.Stat.Position,
                   fEngValue => #fDummy);
END_REGION

REGION Network 78: HBL_PT_701 Filter dryer suction pressure
   "fcAnalogInput"(bValidData := "RIO2_Slot6_I".CH01_ok,
                   iAI := "RIO2_Slot6_I".CH01,
                   fOffset := "DB_System".BarometricOffset,
                   sTag := "DB_AI".HBL_PT_701,
                   fEngValue => #fDummy);
END_REGION

REGION Network 79: HBL_PT_702 Filter dryer discharge pressure
   "fcAnalogInput"(bValidData := "RIO2_Slot6_I".CH02_ok,
                   iAI := "RIO2_Slot6_I".CH02,
                   fOffset := "DB_System".BarometricOffset,
                   sTag := "DB_AI".HBL_PT_702,
                   fEngValue => #fDummy);
END_REGION

REGION Network 80: HBL_PT_703 Filter dryer differential pressure
   // PT703 = PT701 - PT702 (Pressure drop)
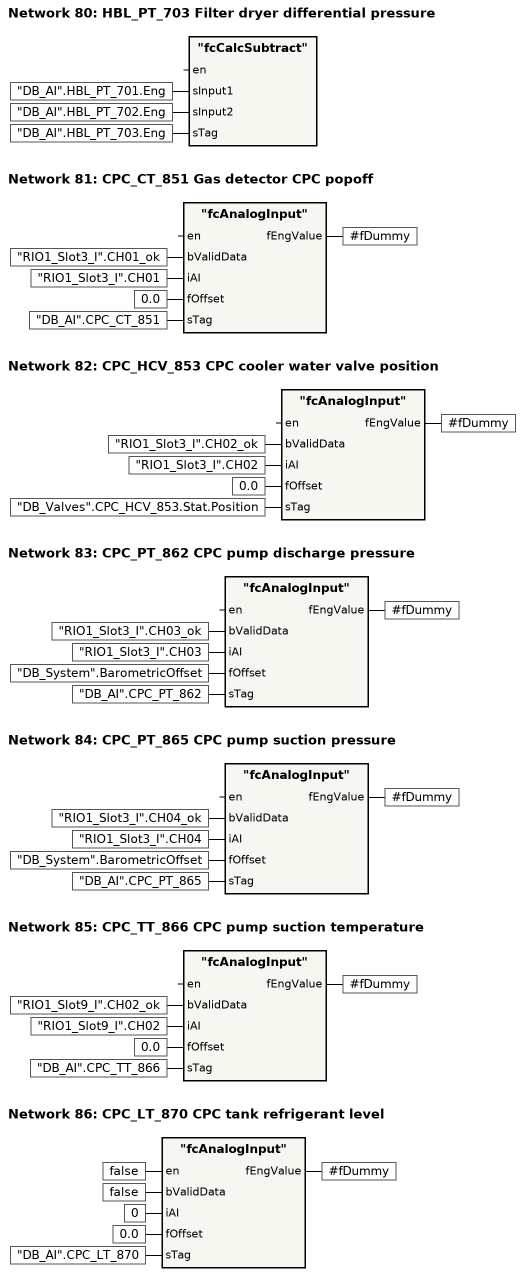
   "fcCalcSubtract"(sInput1 := "DB_AI".HBL_PT_701.Eng,
                    sInput2 := "DB_AI".HBL_PT_702.Eng,
                    sTag := "DB_AI".HBL_PT_703.Eng);
END_REGION

REGION Network 81: CPC_CT_851 Gas detector CPC popoff
   "fcAnalogInput"(bValidData := "RIO1_Slot3_I".CH01_ok,
                   iAI := "RIO1_Slot3_I".CH01,
                   fOffset := 0.0,
                   sTag := "DB_AI".CPC_CT_851,
                   fEngValue => #fDummy);
END_REGION

REGION Network 82: CPC_HCV_853 CPC cooler water valve position
   "fcAnalogInput"(bValidData := "RIO1_Slot3_I".CH02_ok,
                   iAI := "RIO1_Slot3_I".CH02,
                   fOffset := 0.0,
                   sTag := "DB_Valves".CPC_HCV_853.Stat.Position,
                   fEngValue => #fDummy);
END_REGION

REGION Network 83: CPC_PT_862 CPC pump discharge pressure
   "fcAnalogInput"(bValidData := "RIO1_Slot3_I".CH03_ok,
                   iAI := "RIO1_Slot3_I".CH03,
                   fOffset := "DB_System".BarometricOffset,
                   sTag := "DB_AI".CPC_PT_862,
                   fEngValue => #fDummy);
END_REGION

REGION Network 84: CPC_PT_865 CPC pump suction pressure
   "fcAnalogInput"(bValidData := "RIO1_Slot3_I".CH04_ok,
                   iAI := "RIO1_Slot3_I".CH04,
                   fOffset := "DB_System".BarometricOffset,
                   sTag := "DB_AI".CPC_PT_865,
                   fEngValue => #fDummy);
END_REGION

REGION Network 85: CPC_TT_866 CPC pump suction temperature
   "fcAnalogInput"(bValidData := "RIO1_Slot9_I".CH02_ok,
                   iAI := "RIO1_Slot9_I".CH02,
                   fOffset := 0.0,
                   sTag := "DB_AI".CPC_TT_866,
                   fEngValue => #fDummy);
END_REGION

REGION Network 86: CPC_LT_870 CPC tank refrigerant level
   IF false THEN
       "fcAnalogInput"(bValidData := false,
                       iAI := 0,
                       fOffset := 0.0,
                       sTag := "DB_AI".CPC_LT_870,
                       fEngValue => #fDummy);
   END_IF;
END_REGION

REGION Network 87: CPC_TT_871 CPC tank refrigerant temperature
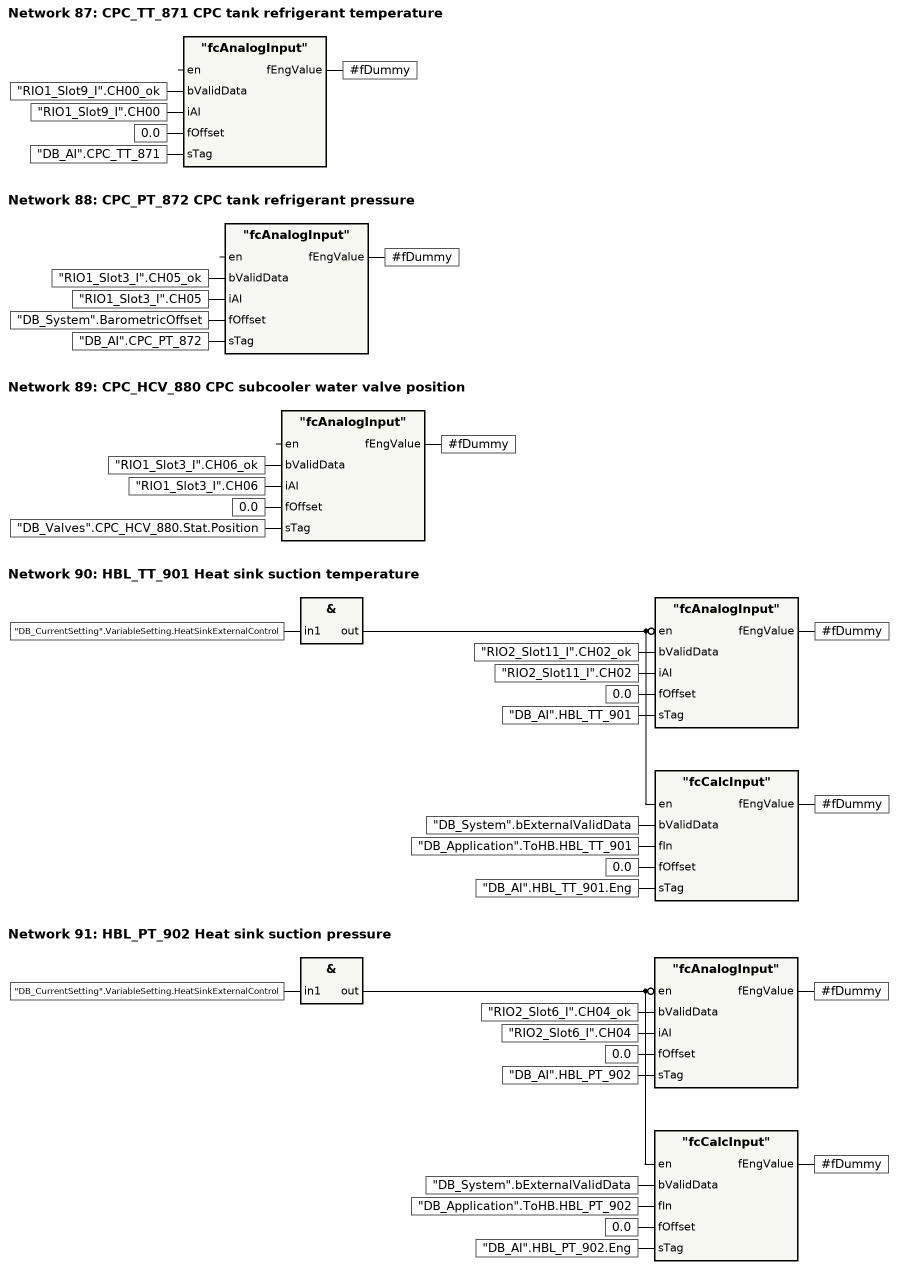
   "fcAnalogInput"(bValidData := "RIO1_Slot9_I".CH00_ok,
                   iAI := "RIO1_Slot9_I".CH00,
                   fOffset := 0.0,
                   sTag := "DB_AI".CPC_TT_871,
                   fEngValue => #fDummy);
END_REGION

REGION Network 88: CPC_PT_872 CPC tank refrigerant pressure
   "fcAnalogInput"(bValidData := "RIO1_Slot3_I".CH05_ok,
                   iAI := "RIO1_Slot3_I".CH05,
                   fOffset := "DB_System".BarometricOffset,
                   sTag := "DB_AI".CPC_PT_872,
                   fEngValue => #fDummy);
END_REGION

REGION Network 89: CPC_HCV_880 CPC subcooler water valve position
   "fcAnalogInput"(bValidData := "RIO1_Slot3_I".CH06_ok,
                   iAI := "RIO1_Slot3_I".CH06,
                   fOffset := 0.0,
                   sTag := "DB_Valves".CPC_HCV_880.Stat.Position,
                   fEngValue => #fDummy);
END_REGION

REGION Network 90: HBL_TT_901 Heat sink suction temperature
   #_w1 := "DB_CurrentSetting".VariableSetting.HeatSinkExternalControl;
   IF NOT "DB_CurrentSetting".VariableSetting.HeatSinkExternalControl THEN
       "fcAnalogInput"(bValidData := "RIO2_Slot11_I".CH02_ok,
                       iAI := "RIO2_Slot11_I".CH02,
                       fOffset := 0.0,
                       sTag := "DB_AI".HBL_TT_901,
                       fEngValue => #fDummy);
   END_IF;
   IF #_w1 THEN
       "fcCalcInput"(bValidData := "DB_System".bExternalValidData,
                     fIn := "DB_Application".ToHB.HBL_TT_901,
                     fOffset := 0.0,
                     sTag := "DB_AI".HBL_TT_901.Eng,
                     fEngValue => #fDummy);
   END_IF;
END_REGION

REGION Network 91: HBL_PT_902 Heat sink suction pressure
   #_w1 := "DB_CurrentSetting".VariableSetting.HeatSinkExternalControl;
   IF NOT "DB_CurrentSetting".VariableSetting.HeatSinkExternalControl THEN
       "fcAnalogInput"(bValidData := "RIO2_Slot6_I".CH04_ok,
                       iAI := "RIO2_Slot6_I".CH04,
                       fOffset := 0.0,
                       sTag := "DB_AI".HBL_PT_902,
                       fEngValue => #fDummy);
   END_IF;
   IF #_w1 THEN
       "fcCalcInput"(bValidData := "DB_System".bExternalValidData,
                     fIn := "DB_Application".ToHB.HBL_PT_902,
                     fOffset := 0.0,
                     sTag := "DB_AI".HBL_PT_902.Eng,
                     fEngValue => #fDummy);
   END_IF;
END_REGION

REGION Network 92: HBL_CT_950 Gas detector container/compressor room
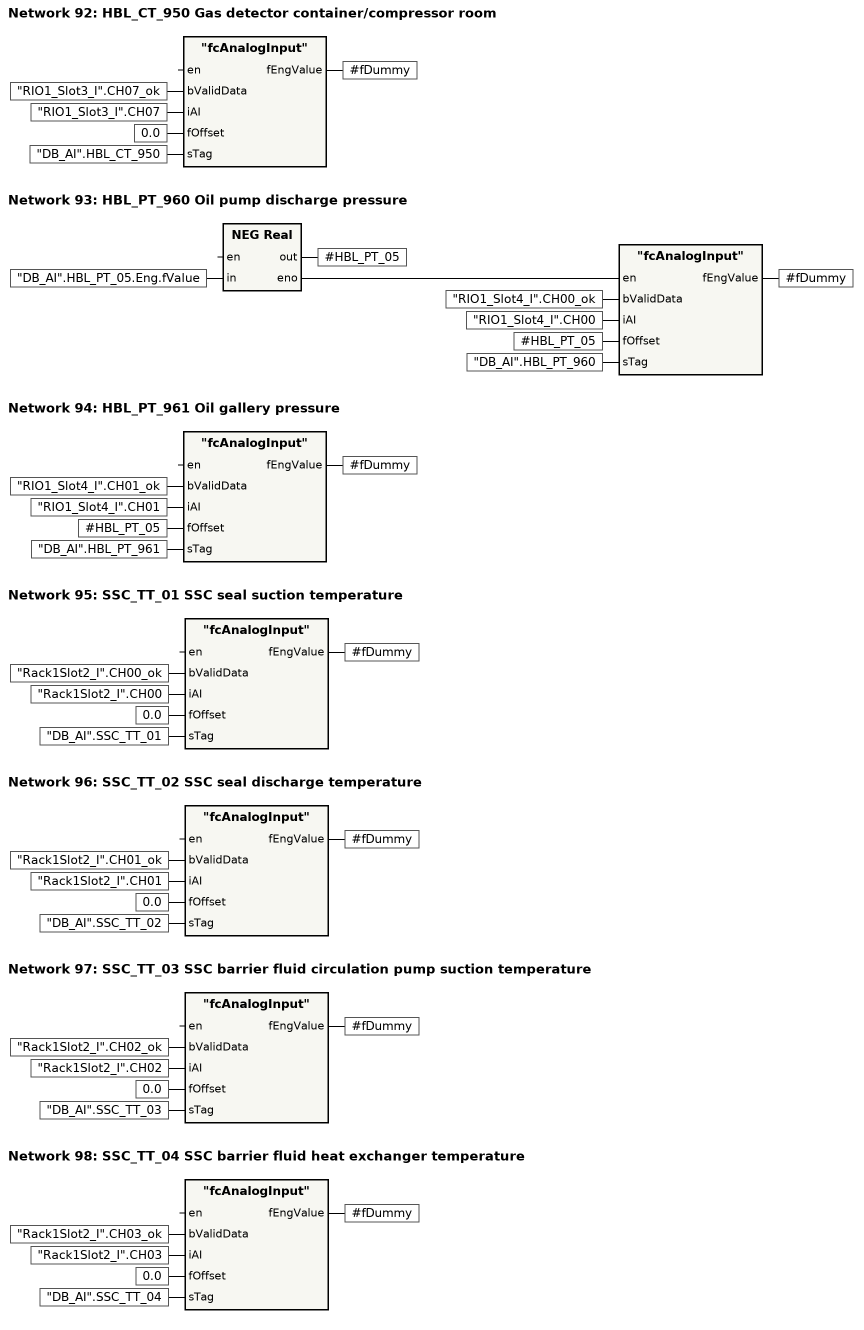
   "fcAnalogInput"(bValidData := "RIO1_Slot3_I".CH07_ok,
                   iAI := "RIO1_Slot3_I".CH07,
                   fOffset := 0.0,
                   sTag := "DB_AI".HBL_CT_950,
                   fEngValue => #fDummy);
END_REGION

REGION Network 93: HBL_PT_960 Oil pump discharge pressure
   // Relative to the crankcase pressure
   #HBL_PT_05 := -"DB_AI".HBL_PT_05.Eng.fValue;
   "fcAnalogInput"(bValidData := "RIO1_Slot4_I".CH00_ok,
                   iAI := "RIO1_Slot4_I".CH00,
                   fOffset := #HBL_PT_05,
                   sTag := "DB_AI".HBL_PT_960,
                   fEngValue => #fDummy);
END_REGION

REGION Network 94: HBL_PT_961 Oil gallery pressure
   // Relative to the crankcase pressure
   "fcAnalogInput"(bValidData := "RIO1_Slot4_I".CH01_ok,
                   iAI := "RIO1_Slot4_I".CH01,
                   fOffset := #HBL_PT_05,
                   sTag := "DB_AI".HBL_PT_961,
                   fEngValue => #fDummy);
END_REGION

REGION Network 95: SSC_TT_01 SSC seal suction temperature
   "fcAnalogInput"(bValidData := "Rack1Slot2_I".CH00_ok,
                   iAI := "Rack1Slot2_I".CH00,
                   fOffset := 0.0,
                   sTag := "DB_AI".SSC_TT_01,
                   fEngValue => #fDummy);
END_REGION

REGION Network 96: SSC_TT_02 SSC seal discharge temperature
   "fcAnalogInput"(bValidData := "Rack1Slot2_I".CH01_ok,
                   iAI := "Rack1Slot2_I".CH01,
                   fOffset := 0.0,
                   sTag := "DB_AI".SSC_TT_02,
                   fEngValue => #fDummy);
END_REGION

REGION Network 97: SSC_TT_03 SSC barrier fluid circulation pump suction temperature
   "fcAnalogInput"(bValidData := "Rack1Slot2_I".CH02_ok,
                   iAI := "Rack1Slot2_I".CH02,
                   fOffset := 0.0,
                   sTag := "DB_AI".SSC_TT_03,
                   fEngValue => #fDummy);
END_REGION

REGION Network 98: SSC_TT_04 SSC barrier fluid heat exchanger temperature
   "fcAnalogInput"(bValidData := "Rack1Slot2_I".CH03_ok,
                   iAI := "Rack1Slot2_I".CH03,
                   fOffset := 0.0,
                   sTag := "DB_AI".SSC_TT_04,
                   fEngValue => #fDummy);
END_REGION

REGION Network 99: SSC_PIT_01 SSC barrier fluid accumulator pressure
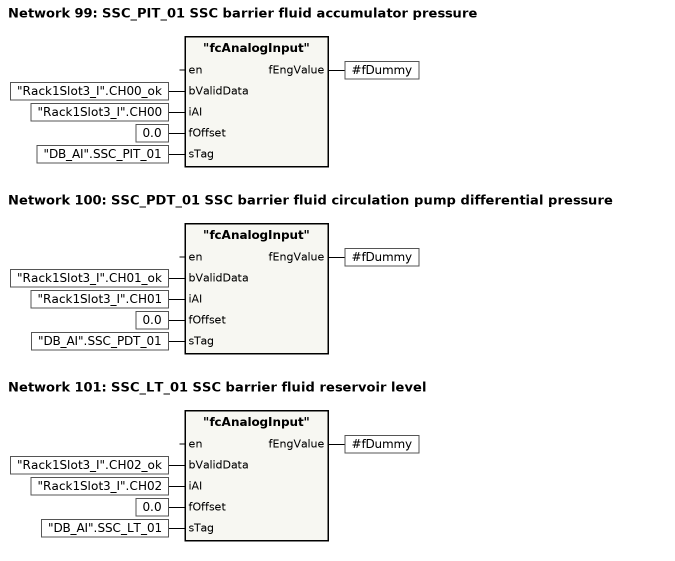
   "fcAnalogInput"(bValidData := "Rack1Slot3_I".CH00_ok,
                   iAI := "Rack1Slot3_I".CH00,
                   fOffset := 0.0,
                   sTag := "DB_AI".SSC_PIT_01,
                   fEngValue => #fDummy);
END_REGION

REGION Network 100: SSC_PDT_01 SSC barrier fluid circulation pump differential pressure
   "fcAnalogInput"(bValidData := "Rack1Slot3_I".CH01_ok,
                   iAI := "Rack1Slot3_I".CH01,
                   fOffset := 0.0,
                   sTag := "DB_AI".SSC_PDT_01,
                   fEngValue => #fDummy);
END_REGION

REGION Network 101: SSC_LT_01 SSC barrier fluid reservoir level
   "fcAnalogInput"(bValidData := "Rack1Slot3_I".CH02_ok,
                   iAI := "Rack1Slot3_I".CH02,
                   fOffset := 0.0,
                   sTag := "DB_AI".SSC_LT_01,
                   fEngValue => #fDummy);
END_REGION
END_FUNCTION_BLOCK
